PROGRAM MAIN
VAR
END_VAR

END_PROGRAM

(* stored: Version 1.1.0.1, ProductVersion 3.1.0.36
   POU MAIN: Id {5923f2dc-4fa6-4fd3-b2cd-d0af9d26a14f} *)
